2970:  !PR[57] assitant Unloading preses ;
2971:  CALL CREATE_PR(57,(-133.703),92.431,364.782,167.802,(-88.383),(-166.755)) ;
2972:  !PR[58] assitant Unloading preses ;
2973:  CALL CREATE_PR(58,(-133.703),92.431,364.782,167.804,(-88.383),(-166.755)) ;
2974:  ENDIF ;
2975:   ;
2976:  !---------------------------- ;
2977:  !SR[2] = "JOB_VAR_OD_GRIP" ;
2978:  !JOB_VAR_COMMON(R[103])'s value ;
2979:  !---------------------------- ;
2980:  !2By3 SR[2] INF, Max 18(Straight) ;
2981:  !R[103]=200 ;
2982:  !2By3 INF 45 Degree Diagonal Shif ;
2983:  !R[103]=210 ;
2984:  !---------------------------- ;
2985:  !3By4 SR[2] INF, Max 36(Straight) ;
2986:  !R[103]=250 ;
2987:  !3By4 INF 45 Degree Diagonal Shif ;
2988:  !R[103]=260 ;
2989:  !---------------------------- ;
2990:  !R[103] "JOB_PROFILE" Selection ;
2991:  R[103]=200    ;
2992:  CALL JOB_VAR_COMMON(R[103]) ;
2993:   ;
2994:  ENDIF ;
2995:   ;
2996:  JMP LBL[9999] ;
2997:   ;
2998:  !Job 102779700 Logic Ends ;
2999:  !--------------------------- ;
3000:   ;
3001:  LBL[9814] ;
3002:  !--------------------------- ;
3003:  !Rapid Ball ;
3004:  !Item 102649814 , Rev xxx ;
3005:  !Last Modified: 2021-08-26 ;
3006:  !Modified by: Tsuu ;
3007:  !2.0 IN Height ;
3008:  !0 ID, 2.0 OD ;
3009:  !OD Jaw #3001 ;
3010:  !--------------------------- ;
3011:  IF (R[70]=9814) THEN ;
3012:  !Define Parameters for INF/OTF ;
3013:  !R[105]=AR[1]=100, 2By3 Sheet ;
3014:  !R[105]=AR[1]=200, 3By4 Sheet ;
3015:  !R[105]=AR[1]=300, 5By7 Sheet ;
3016:  CALL JOB_VAR_SETUP(400) ;
3017:   ;
3018:  !--------------------------- ;
3019:  !Define Parameters for Job ;
3020:  !R[85] "INF_JAW_OFFSET"(Hgt) ;
3021:  R[85]=97    ;
3022:  !R[86] "INF_PICK_OFFSET" 50mm/sec ;
3023:  R[86]=0    ;
3024:  !R[87] "MAIN_LOAD_OFFSET" (PRELOA ;
3025:  R[87]=100    ;
3026:  !R[100] "GRIPPER_ID" 3 values ;
3027:  !If =100, ID Grippers Installed ;
3028:  !If =200, OD Grippers Installed ;
3029:  !If =300, OD 45 Degree Grippers ;
3030:  R[100]=200    ;
3031:  !--------------------------- ;
3032:   ;
3033:  !If using previous setup data ;
3034:  IF (R[71]=9814) THEN ;
3035:   ;
3036:  !--------------------------- ;
3037:  !1st: Height of Raw piece ;
3038:  R[190]=56.15    ;
3039:  !2nd: Height of Finish piece ;
3040:  R[191]=50    ;
3041:  !3rd: Infeed Height Offset ;
3042:  R[192]=(-98)    ;
3043:  !4th: Outfeed Height Offset ;
3044:  R[193]=(-46.5)    ;
3045:  !--------------------------- ;
3046:   ;
3047:  CALL CREATE_REG(R[190],R[191],R[192],R[193]) ;
3048:   ;
3049:  ENDIF ;
3050:   ;
3051:  !If new loading or offloading pos ;
3052:  !SET R[104] "IMPORT_LOADPOS" ;
3053:  !SET R[104]=1000, Otherwise NO ;
3054:  R[104]=1000    ;
3055:  IF (R[104]=1000) THEN ;
3056:  !R[260]=43, Preload Pos1 ;
3057:  !R[270]=44, Preload PosFinal ;
3058:  !R[300]=53, Offload PosFinal ;
3059:  !PR[43] Pre-Loading Pos1 ;
3060:  CALL CREATE_PR(43,168.835,(-63.534),347.629,158.268,89.347,156.235) ;
3061:  !PR[44] Final Loading Position ;
3062:  CALL CREATE_PR(44,168.927,(-63.781),356.006,158.173,89.348,156.13) ;
3063:  !PR[53] Pre Unloading Position ;
3064:  CALL CREATE_PR(53,(-129.883),93.702,179.02,170.509,(-88.382),(-168.991)) ;
3065:  !PR[54] Final Unloading Position ;
3066:  CALL CREATE_PR(54,(-128.536),94.044,130.257,170.547,(-88.382),(-169.034)) ;
3067:  !PR[56] assitant Unloading preses ;
3068:  CALL CREATE_PR(56,(-131.536),105.713,233.177,173.746,(-88.233),(-175.647)) ;
3069:  !PR[57] assitant Unloading preses ;
3070:  CALL CREATE_PR(57,(-131.536),105.713,233.177,173.746,(-88.233),(-175.647)) ;
3071:  !PR[58] assitant Unloading preses ;
3072:  CALL CREATE_PR(58,(-131.536),105.713,233.177,173.746,(-88.233),(-175.647)) ;
3073:  ENDIF ;
3074:   ;
3075:  !---------------------------- ;
3076:  !SR[2] = "JOB_VAR_OD_GRIP" ;
3077:  !JOB_VAR_COMMON(R[103])'s value ;
3078:  !---------------------------- ;
3079:  !2By3 SR[2] INF, Max 18(Straight) ;
3080:  !R[103]=200 ;
3081:  !2By3 INF 45 Degree Diagonal Shif ;
3082:  !R[103]=210 ;
3083:  !---------------------------- ;
3084:  !3By4 SR[2] INF, Max 36(Straight) ;
3085:  !R[103]=250 ;
3086:  !3By4 INF 45 Degree Diagonal Shif ;
3087:  !R[103]=260 ;
3088:  !---------------------------- ;
3089:  !R[103] "JOB_PROFILE" Selection ;
3090:  R[103]=270    ;
3091:  CALL JOB_VAR_COMMON(R[103]) ;
3092:   ;
3093:  ENDIF ;
3094:   ;
3095:  JMP LBL[9999] ;
3096:   ;
3097:  !Job 102649814 Logic Ends ;
3098:  !--------------------------- ;
3099:   ;
3100:  LBL[9990] ;
3101:  !--------------------------- ;
3102:  !KAREL PROGRAM ;
3103:  !Item 1111199990  ;
3104:  !Last Modified: 2026-Sep-17 ;
3105:  !Modified by: Erfan ;
3106:  !--------------------------- ;
3107:  IF (R[70]=9990) THEN ;
3108:  !Define Parameters for INF/OTF ;
3109:  !R[105]=AR[1]=100, 2By3 Sheet ;
3110:  !R[105]=AR[1]=200, 3By4 Sheet ;
3111:  !R[105]=AR[1]=300, 5By7 Sheet ;
3112:  CALL JOB_VAR_SETUP(400) ;
3113:  CALL GN_CLS_SC_F9 ;
3114:  MESSAGE[OD GRIPPING STARTS] ;
3115:  WAIT 3.00(sec) ;
3116:   ;
3117:  !--------------------------- ;
3118:  !Define Parameters for Job ;
3119:  !R[85] "INF_JAW_OFFSET"(Hgt) ;
3120:  R[85]=97    ;
3121:  !R[86] "INF_PICK_OFFSET" 50mm/sec ;
3122:  R[86]=0    ;
3123:  !R[87] "MAIN_LOAD_OFFSET" (PRELOA ;
3124:  R[87]=100    ;
3125:  !R[100] "GRIPPER_ID" 3 values ;
3126:  !If =100, ID Grippers Installed ;
3127:  !If =200, OD Grippers Installed ;
3128:  !If =300, OD 45 Degree Grippers ;
3129:  R[100]=200    ;
3130:  !--------------------------- ;
3131:   ;
3132:  !If using previous setup data ;
3133:  IF (R[71]=9990) THEN ;
3134:   ;
3135:  !--------------------------- ;
3136:  !1st: Height of Raw piece ;
3137:  R[190]=56.15    ;
3138:  !2nd: Height of Finish piece ;
3139:  R[191]=50    ;
3140:  !3rd: Infeed Height Offset ;
3141:  R[192]=(-98)    ;
3142:  !4th: Outfeed Height Offset ;
3143:  R[193]=(-46.5)    ;
3144:  !--------------------------- ;
3145:   ;
3146:  CALL CREATE_REG(R[190],R[191],R[192],R[193]) ;
3147:   ;
3148:  ENDIF ;
3149:   ;
3150:  !If new loading or offloading pos ;
3151:  !SET R[104] "IMPORT_LOADPOS" ;
3152:  !SET R[104]=1000, Otherwise NO ;
3153:  R[104]=1000    ;
3154:  IF (R[104]=1000) THEN ;
3155:  !R[260]=43, Preload Pos1 ;
3156:  !R[270]=44, Preload PosFinal ;
3157:  !R[300]=53, Offload PosFinal ;
3158:  !PR[43] Pre-Loading Pos1 ;
3159:  CALL CREATE_PR(43,168.835,(-63.534),347.629,158.268,89.347,156.235) ;
3160:  !PR[44] Final Loading Position ;
3161:  CALL CREATE_PR(44,168.927,(-63.781),356.006,158.173,89.348,156.13) ;
3162:  !PR[53] Pre Unloading Position ;
3163:  CALL CREATE_PR(53,(-129.883),93.702,179.02,170.509,(-88.382),(-168.991)) ;
3164:  !PR[54] Final Unloading Position ;
3165:  CALL CREATE_PR(54,(-128.536),94.044,130.257,170.547,(-88.382),(-169.034)) ;
3166:  !PR[56] assitant Unloading preses ;
3167:  CALL CREATE_PR(56,(-131.536),105.713,233.177,173.746,(-88.233),(-175.647)) ;
3168:  !PR[57] assitant Unloading preses ;
3169:  CALL CREATE_PR(57,(-131.536),105.713,233.177,173.746,(-88.233),(-175.647)) ;
3170:  !PR[58] assitant Unloading preses ;
3171:  CALL CREATE_PR(58,(-131.536),105.713,233.177,173.746,(-88.233),(-175.647)) ;
3172:  ENDIF ;
3173:   ;
3174:  !---------------------------- ;
3175:  !SR[2] = "JOB_VAR_OD_GRIP" ;
3176:  !JOB_VAR_COMMON(R[103])'s value ;
3177:  !---------------------------- ;
3178:  !2By3 SR[2] INF, Max 18(Straight) ;
3179:  !R[103]=200 ;
3180:  !2By3 INF 45 Degree Diagonal Shif ;
3181:  !R[103]=210 ;
3182:  !---------------------------- ;
3183:  !3By4 SR[2] INF, Max 36(Straight) ;
3184:  !R[103]=250 ;
3185:  !3By4 INF 45 Degree Diagonal Shif ;
3186:  !R[103]=260 ;
3187:  !---------------------------- ;
3188:  !R[103] "JOB_PROFILE" Selection ;
3189:  R[103]=270    ;
3190:  CALL JOB_VAR_COMMON(R[103]) ;
3191:   ;
3192:  ENDIF ;
3193:   ;
3194:  JMP LBL[9999] ;
3195:   ;
3196:  !Job 102649814 Logic Ends ;
3197:  !--------------------------- ;
3198:   ;
3199:  LBL[9999] ;
3200:  !Program Ends, no further logic ;
3201:  END ;
/POS
/END
